FUNCTION_BLOCK Test_TEvent_AddEventHandler_IncsNumberOfEventHandlers EXTENDS TUnitTestbase
VAR
    TestEvent : TTestEvent;
    TestEventHandler : TTestEventHandler;
END_VAR



TestEvent
    .ClearEventHandlers()
    .AddEventHandler(TestEventHandler);
    
Assertion.AssertEquals_UDINT(
    Expected := 1,
    Actual   := TestEvent.EventHandlers.Count,
    ObjectName := _TestName,
    VariableName  := 'TestEvent.EventHandlers.Count');
    

TestFinished();

END_FUNCTION_BLOCK

(* stored: Version 1.1.0.1, ProductVersion 3.1.4024.4
   POU Test_TEvent_AddEventHandler_IncsNumberOfEventHandlers: Id {eda56f75-f01d-4e29-8f23-82687b9fbdd7}, SpecialFunc None *)
